FUNCTION_BLOCK Homing_Mode
VAR_INPUT
	NodeID				: BYTE; (* This Port No. addresses the CANopen Node (see System Manager) *)
	Start 				: BOOL;
	Current_State 		: E_Statemachine_State;	
	Statusword			: WORD;	
	Homing_parameters	: ST_Homing_parameters;
END_VAR
VAR_OUTPUT
	Controlword 		: WORD;
	Mode_of_operation 	: E_Mode_of_operation	:= E_Mode_of_operation.No_mode_active;
	Finished			: BOOL;
END_VAR
VAR
	Index 			: BYTE := 0;
	
	SDO_WRITE		: FB_SDO_WRITE;
	WriteData		: ARRAY [0..255] OF BYTE;
	
	SDO_READ		: FB_SDO_READ;
	ReadStart		: BOOL;
	ReadError		: DWORD;
	ReadData		: ARRAY [0..255] OF BYTE;
	
	fbTonDelay		: TON;
	Start_old		: BOOL := FALSE;
END_VAR

// Restart after complete run
IF NOT Start_old AND Start THEN
	Index := 0;
	Finished := FALSE;
END_IF


CASE Index OF	
	0: // Switch to state 'Switch on disabled'
		IF (Start) THEN
			Mode_of_operation := E_Mode_of_operation.No_mode_active;
			Controlword := CONTROLWORD_STATE_CHANGE(Current_State, E_Statemachine_State.Switch_on_disabled);
			IF (Current_State = E_Statemachine_State.Switch_on_disabled) THEN			
				Index := Index + 2;
			ELSE
				Index := Index + 1;		
			END_IF
		END_IF
		
			
	1: // Wait for 'Switch on disabled'
		Controlword := CONTROLWORD_STATE_CHANGE(Current_State, E_Statemachine_State.Switch_on_disabled);	
		IF (Current_State = E_Statemachine_State.Switch_on_disabled) THEN			
			Index := Index + 1;		
		END_IF
					
		
	2: // Set Mode of operation
		Mode_of_operation := E_Mode_of_operation.Homing_mode;	
		Controlword := CONTROLWORD_STATE_CHANGE(Current_State, E_Statemachine_State.Switch_on_disabled);				
		IF (PDO.Mode_of_operation_display = E_Mode_of_operation.Homing_mode) THEN			
			IF Homing_parameters.Homing_mode = E_Homing_mode.Homing_on_current_position THEN
				Index := Index + 1 + 3*2;
			ELSE
				Index := Index + 1;		
			END_IF
		END_IF

		
	3: // Set Speed during search for switch		
		Controlword := CONTROLWORD_STATE_CHANGE(Current_State, E_Statemachine_State.Switch_on_disabled);	
		WriteData[0] := DWORD_TO_BYTE(Homing_parameters.Speed_switch);
		WriteData[1] := DWORD_TO_BYTE(SHR(Homing_parameters.Speed_switch,8));
		WriteData[2] := DWORD_TO_BYTE(SHR(Homing_parameters.Speed_switch,16));
		WriteData[3] := DWORD_TO_BYTE(SHR(Homing_parameters.Speed_switch,24));	
		SDO_WRITE(	
			AdsNetID		:= GLB.ADSNetID_CAN,
			PortNr			:= 16#1000 + GLB.NodeID,
			CO_Index		:= 16#6099,
			CO_SubIndex		:= 16#01,
			DataLength		:= 4,
			WriteData		:= WriteData,
			StartWriting	:= TRUE	
		);	
		Index := Index + 1;		
		
	4: // Wait for finish sdo transfer	
		Controlword := CONTROLWORD_STATE_CHANGE(Current_State, E_Statemachine_State.Switch_on_disabled);	
		SDO_WRITE(StartWriting := FALSE);
		IF SDO_WRITE.WriteDataFinished THEN
			Index := Index + 1;			
		END_IF	
		
		
	5: // Set Spped during search for zero			
		Controlword := CONTROLWORD_STATE_CHANGE(Current_State, E_Statemachine_State.Switch_on_disabled);	
		WriteData[0] := DWORD_TO_BYTE(Homing_parameters.Speed_zero);
		WriteData[1] := DWORD_TO_BYTE(SHR(Homing_parameters.Speed_zero,8));
		WriteData[2] := DWORD_TO_BYTE(SHR(Homing_parameters.Speed_zero,16));
		WriteData[3] := DWORD_TO_BYTE(SHR(Homing_parameters.Speed_zero,24));	
		SDO_WRITE(	
			AdsNetID		:= GLB.ADSNetID_CAN,
			PortNr			:= 16#1000 + GLB.NodeID,
			CO_Index		:= 16#6099,
			CO_SubIndex		:= 16#02,
			DataLength		:= 4,
			WriteData		:= WriteData,
			StartWriting	:= TRUE	
		);	
		Index := Index + 1;		
		
	6: // Wait for finish sdo transfer	
		Controlword := CONTROLWORD_STATE_CHANGE(Current_State, E_Statemachine_State.Switch_on_disabled);	
		SDO_WRITE(StartWriting := FALSE);
		IF SDO_WRITE.WriteDataFinished THEN
			Index := Index + 1;			
		END_IF		
		
		
	7: // Set Homing acceleration		
		Controlword := CONTROLWORD_STATE_CHANGE(Current_State, E_Statemachine_State.Switch_on_disabled);	
		WriteData[0] := DWORD_TO_BYTE(Homing_parameters.Acceleration);
		WriteData[1] := DWORD_TO_BYTE(SHR(Homing_parameters.Acceleration,8));
		WriteData[2] := DWORD_TO_BYTE(SHR(Homing_parameters.Acceleration,16));
		WriteData[3] := DWORD_TO_BYTE(SHR(Homing_parameters.Acceleration,24));	
		SDO_WRITE(	
			AdsNetID		:= GLB.ADSNetID_CAN,
			PortNr			:= 16#1000 + GLB.NodeID,
			CO_Index		:= 16#609A,
			CO_SubIndex		:= 16#00,
			DataLength		:= 4,
			WriteData		:= WriteData,
			StartWriting	:= TRUE	
		);	
		Index := Index + 1;		
		
	8: // Wait for finish sdo transfer	
		Controlword := CONTROLWORD_STATE_CHANGE(Current_State, E_Statemachine_State.Switch_on_disabled);	
		SDO_WRITE(StartWriting := FALSE);
		IF SDO_WRITE.WriteDataFinished THEN
			Index := Index + 1;			
		END_IF	
		
		
	9: // Set Homing mode		
		Controlword := CONTROLWORD_STATE_CHANGE(Current_State, E_Statemachine_State.Switch_on_disabled);	
		WriteData[0] := Homing_parameters.Homing_mode;
		SDO_WRITE(	
			AdsNetID		:= GLB.ADSNetID_CAN,
			PortNr			:= 16#1000 + GLB.NodeID,
			CO_Index		:= 16#6098,
			CO_SubIndex		:= 16#00,
			DataLength		:= 1,
			WriteData		:= WriteData,
			StartWriting	:= TRUE	
		);	
		Index := Index + 1;		
		
	10: // Wait for finish sdo transfer	
		Controlword := CONTROLWORD_STATE_CHANGE(Current_State, E_Statemachine_State.Switch_on_disabled);	
		SDO_WRITE(StartWriting := FALSE);
		IF SDO_WRITE.WriteDataFinished THEN
			Index := Index + 1;			
		END_IF		
		
		
	11: // Switch State to 'Operation enabled'
		Controlword := CONTROLWORD_STATE_CHANGE(Current_State, E_Statemachine_State.Operation_enabled);		
		IF (Current_State = E_Statemachine_State.Operation_enabled) THEN			
			Index := Index + 1;
		END_IF
		
		
	12: // Start homing and wait for finish
		Controlword := 16#1F;		
		IF (Statusword AND E_Statusword_Bits.HM_Homing_attained) <> 0 THEN			
			Index := Index + 1;		
		END_IF
	
		
	13: // Switch State to 'Switch on disabled'
		Controlword := CONTROLWORD_STATE_CHANGE(Current_State, E_Statemachine_State.Switch_on_disabled);	
		IF Current_State = E_Statemachine_State.Switch_on_disabled THEN			
			Index := 255;
		END_IF
		
		
	255: // Finished 
		Controlword := CONTROLWORD_STATE_CHANGE(Current_State, E_Statemachine_State.Switch_on_disabled);	
		FINISHED := TRUE;
				
		
	ELSE
		Index := 255;
			
END_CASE


Start_old := Start;

END_FUNCTION_BLOCK

(* stored: Version 1.1.0.1, ProductVersion 3.1.4024.11
   POU Homing_Mode: Id {ccc83746-f290-45c8-8130-00bcc4c808c0}, SpecialFunc None *)
